FUNCTION_BLOCK FB_MoveRegister4
VAR_INPUT
	bFirstCycle	:BOOL;						//Bit od pierwszego cyklu, żeby nie wykrywało zbocza opadającego
	bTrigger	:BOOL;						// BIt do wyzwalania przesuniecia o 4
	tTriggerFilterTimeOn	:TIME:=T#0MS;	// Czas filtrowania wejścia Trigger na załączenie
	tTriggerFilterTimeOFF	:TIME:=T#0MS;	// Czas filtorwania wejścia Trigger na wyłaczenie
	bInvertWriting: BOOL;					//Bit zapisu w odwrotenj kolejnosci
	bTriggerBottle	:BOOL;					// Zapisywanie czy butelka jest czy nie ( jeżeli jest włączona kontrola obecności)
	iEntrenceArrayElements	:UINT;			// Licznik ilości elementów w tablicy wejściowej
	iExitArrayElements	:UINT;				// Licznik ilosco elementów w tablicy wyjściowej
	bWithFormControlTrigerCounter	:BOOL;	// Jezeli na tr
	bMoveOnlyIfFormPresent	:BOOL;			//Przesuwanie tylko jeśli jest obecna formatka
	bMoveOnlyToLastExitRegister	:BOOL;		// PRzesuniecie tylko na ostatni rejstr wyjsciowy
	bMoveOnlyToLastRegister: BOOL;
	bNoKeepTryingMove: BOOL; 				//PRóbuj dakej przesunać jeżelei nie ma miejsca
	bReset	:BOOL;							// Czyszczenie tablicy
	eClearPackageState	:S_PackageState;	//Deklaracja czystego rejestru
	
	
	bRotateEntranceRegisterBefore: BOOL;	//Przesuwanie rejestrru wejściowego, a następnie go obrót
END_VAR
VAR_OUTPUT
	bError	:BOOL;	//Bład w sekwencji
	iError	:INT;	//Numer błędu 
	bTriggerDone :BOOL;		//Przesunięcie wykonane
	bTriggerFilteredOUT:BOOL;	//Sygnał przefiltorwanego bitu aktywacji przesuniecia 
END_VAR
VAR_IN_OUT
	bTriggerCounter	:BOOL;   //Triger do kasowania
	eEntranceState :ARRAY[1..17] OF S_PackageState;		//Tablica wejściowa danych
	eExitState	:ARRAY[1..17] OF S_PackageState;		//Tablica wyjściowa danych
	bKeepTryingMove	:BOOL;	//Próbuj zapisać formatki dalej, aż do zwolnienia miejsca
END_VAR
VAR
	tofTriggerFilterTimeOff: TOF;	//Czasówka do filtrowania wyzwolenia przesuniecia
	tonTriggerFilterTimeOn: TON;	// Czas do filtrowania wyzwolenia przesuniecia
	bTriggerFiltered: BOOL;		//Bit informujacy o przefiltrowaniu wejscai
	bWithBottleControl: BOOL;	// Bit od kontroli butleki
	rtbTrigger: R_TRIG;		//Bit zbocza narastającego przesuniecia formatki
	rtbTriggerBottle: R_TRIG;	// Bit zbocza narastającego butelki
	rtbReset: R_TRIG;
	bWithCapControl: BOOL;		//Bit kontroli obecnosci nasadki
	i: UINT;		//Licznik pętli
	nFormCounter: UINT; //Licznik formatek
	j: UINT;			//Zmienna pomocncza
	r1: UINT;			//Zmienna pomocnicza
	r2: UINT;			//Zmienna pomocnicza

	TimerResetErrors: TON;
	k: UINT;
	bNotEmptyPlace: BOOL;
END_VAR

//Filtrowanie sygnału wejściowego
tofTriggerFilterTimeOff	(IN:=bTrigger, PT:=tTriggerFilterTimeOff);
tonTriggerFilterTimeOn	(IN:=tofTriggerFilterTimeOff.Q, PT:=tTriggerFilterTimeOn);
bTriggerFiltered 		:= tonTriggerFilterTimeOn.Q;
bTriggerFilteredOUT		:= bTriggerFiltered ;

//TRIGI I TIMERY
IF bWithBottleControl THEN
	rtbTrigger 	(CLK := NOT bTriggerFiltered, Q=>);
	rtbTriggerBottle 	(CLK := NOT bTriggerBottle, Q=>);
ELSIF bWithCapControl THEN
	rtbTrigger 	(CLK := NOT bTriggerFiltered, Q=>);
ELSE
	rtbTrigger 	(CLK := bTriggerFiltered, Q=>);
	rtbTriggerBottle 	(CLK := bTriggerBottle, Q=>);
END_IF

rtbReset 	(CLK := bReset, Q=>);
TimerResetErrors (IN:= bError, PT:=T#1000MS, Q=>);

//RESETOWANIE BLEDU
IF TimerResetErrors.Q THEN
	bError := FALSE;
END_IF

bTriggerDone := FALSE;

// PRzesuniecie rejestrów 

IF iEntrenceArrayElements = iExitArrayElements AND  bFirstCycle THEN
	IF rtbTrigger.Q OR bKeepTryingMove THEN
		bTriggerCounter	:=FALSE;
		bKeepTryingMove	:=FALSE;
		bNotEmptyPlace:=FALSE;
		nFormCounter:=0;
		
		eExitState[1]:= eEntranceState[1];
		eExitState[2]:= eEntranceState[2];
		eExitState[3]:= eEntranceState[3];
		eExitState[4]:= eEntranceState[4];
		
		eEntranceState[1]:=eClearPackageState;
		eEntranceState[2]:=eClearPackageState;
		eEntranceState[3]:=eClearPackageState;
		eEntranceState[4]:=eClearPackageState;
		
		END_IF
	END_IF




//CZYSZCZENIE REJESTRU WEJSCIOWEGO
IF rtbReset.Q THEN
	FOR r1 := 1 TO iEntrenceArrayElements DO
		eEntranceState[r1] := eClearPackageState;
	END_FOR
	FOR r2 := 1 TO iExitArrayElements DO
		eExitState[r2] := eClearPackageState;
	END_FOR
	bKeepTryingMove :=FALSE;
	bTriggerDone := FALSE;
	bTriggerCounter := FALSE; 
	nFormCounter := 0;
	//bBottlePresent := bCapPresent := FALSE; 
	bError := FALSE;
	iError := 0;
END_IF

END_FUNCTION_BLOCK

(* stored: Version 1.1.0.1, ProductVersion 3.1.4026.13, FileIdentifier cbaf34665024e1e879aff9df993534c810302588, FileSignature 544f716b82055c7e2375c1ec0dc75e8deec6c01a4cd1cfe674912cbcd4aa37b7af9f768393a461b4d4e48ce85632641c3072a486333b131395c8b7e85c84e089a56b7451bf29129b9559af4b507b21c811873a22bd86e8569897652f2403a2638161876ad5cf4390bef2a760ad7ce57ccc27c922f5bfc4902818014922e6ad192979f95166d8684921b13726ba97847884e4ebec970283aef0837d9f156b9adaccf32e57ca8ee9a4dacece2f001c583c2f2182f0f7e942754722ceda167ca0d40e6e40617c33fb2cb7014cd2948cf944bea88a7965737632a0e00f20b369c85f8ea4ebc6038e24d10d0167515f8cff0683f2de5a258977b4f43888918c52d09a
   POU FB_MoveRegister4: Id {1d1d0891-4376-4d12-b63a-116844b5dd56}, SpecialFunc None *)
